// Mitsubishi GX Works2 project: BookEX3_2 FB   PLC: Q13UDV

TYPE DateTime : STRUCT
  Year : INT;
  Month : INT;
  Day : INT;
  WeekDay : INT;
  iHour : INT;
  iMin : INT;
  iSec : INT;
  ms : INT;
END_STRUCT END_TYPE

TYPE Vector : STRUCT
  axisX : REAL;
  axisY : REAL;
  axisZ : REAL;
END_STRUCT END_TYPE

TYPE WordBit : STRUCT
  Data : DWORD;
  Flag : BOOL;
END_STRUCT END_TYPE

// global labels: Global
VAR_GLOBAL
  bVar0 AT M5000 : BOOL;
  abArray0 AT M5010 : ARRAY [0..49] OF BOOL;
  sStr0 AT D5000 : STRING[199];
  sStr1 AT D5100 : STRING[199];
  sStr2 AT D5200 : STRING[199];
  sStr3 AT D5300 : STRING[199];
  sStr4 AT D5400 : STRING[199];
  sStr5 AT D5500 : STRING[199];
  sStr6 AT D5600 : STRING[199];
  sStr7 AT D5700 : STRING[199];
  sStr8 AT D5800 : STRING[199];
  sStr9 AT D5900 : STRING[199];
  iVar0 AT D4500 : INT;
  iVar1 AT D4501 : INT;
  iVar2 AT D4502 : INT;
  iVar3 AT D4503 : INT;
  iVar4 AT D4504 : INT;
  iVar5 AT D4505 : INT;
  iVar6 AT D4506 : INT;
  iVar7 AT D4507 : INT;
  iVar8 AT D4508 : INT;
  iVar9 AT D4509 : INT;
  dVar0 AT D4510 : DINT;
  dVar1 AT D4512 : DINT;
  dVar2 AT D4514 : DINT;
  dVar3 AT D4516 : DINT;
  dVar4 AT D4518 : DINT;
  dVar5 AT D4520 : DINT;
  dVar6 AT D4522 : DINT;
  dVar7 AT D4524 : DINT;
  dVar8 AT D4526 : DINT;
  dVar9 AT D4528 : DINT;
  wVar0 AT D4530 : WORD;
  wVar1 AT D4531 : WORD;
  wVar2 AT D4532 : WORD;
  wVar3 AT D4533 : WORD;
  wVar4 AT D4534 : WORD;
  wVar5 AT D4535 : WORD;
  wVar6 AT D4536 : WORD;
  wVar7 AT D4537 : WORD;
  wVar8 AT D4538 : WORD;
  wVar9 AT D4539 : WORD;
  dwVar0 AT D4540 : DWORD;
  dwVar1 AT D4542 : DWORD;
  dwVar2 AT D4544 : DWORD;
  dwVar3 AT D4546 : DWORD;
  dwVar4 AT D4548 : DWORD;
  dwVar5 AT D4550 : DWORD;
  dwVar6 AT D4552 : DWORD;
  dwVar7 AT D4554 : DWORD;
  dwVar8 AT D4556 : DWORD;
  dwVar9 AT D4558 : DWORD;
  fsVar0 AT D4560 : REAL;
  fsVar1 AT D4562 : REAL;
  fsVar2 AT D4564 : REAL;
  fsVar3 AT D4566 : REAL;
  fsVar4 AT D4568 : REAL;
  fsVar5 AT D4570 : REAL;
  fsVar6 AT D4572 : REAL;
  fsVar7 AT D4574 : REAL;
  fsVar8 AT D4576 : REAL;
  fsVar9 AT D4578 : REAL;
  fdVar0 AT D4580 : LREAL;
  tTime0 AT D4620 : TIME;
  tTime1 AT D4622 : TIME;
  tTime2 AT D4624 : TIME;
  tTime3 AT D4626 : TIME;
  tTime4 AT D4628 : TIME;
  tTime5 AT D4630 : TIME;
  tTime6 AT D4632 : TIME;
  tTime7 AT D4634 : TIME;
  tTime8 AT D4636 : TIME;
  tTime9 AT D4638 : TIME;
  tTime10 AT D4640 : TIME;
  bVar1 AT M5001 : BOOL;
  bVar2 AT M5002 : BOOL;
  bVar3 AT M5003 : BOOL;
  bVar4 AT M5004 : BOOL;
  bVar5 AT M5005 : BOOL;
  bVar6 AT M5006 : BOOL;
  bVar7 AT M5007 : BOOL;
  bVar8 AT M5008 : BOOL;
  bVar9 AT M5009 : BOOL;
  abArray1 AT M5060 : ARRAY [0..49] OF BOOL;
  abArray2 AT M5110 : ARRAY [0..49] OF BOOL;
  abArray3 AT M5160 : ARRAY [0..49] OF BOOL;
  abArray4 AT M5210 : ARRAY [0..49] OF BOOL;
  abArray5 AT M5260 : ARRAY [0..49] OF BOOL;
  abArray6 AT M5310 : ARRAY [0..49] OF BOOL;
  abArray7 AT M5360 : ARRAY [0..49] OF BOOL;
  abArray8 AT M5410 : ARRAY [0..49] OF BOOL;
  abArray9 AT M5460 : ARRAY [0..49] OF BOOL;
  fdVar1 AT D4584 : LREAL;
  fdVar2 AT D4588 : LREAL;
  fdVar3 AT D4592 : LREAL;
  fdVar4 AT D4596 : LREAL;
  fdVar5 AT D4600 : LREAL;
  fdVar6 AT D4604 : LREAL;
  fdVar7 AT D4608 : LREAL;
  fdVar8 AT D4612 : LREAL;
  fdVar9 AT D4616 : LREAL;
  afsPen0 AT D2000 : ARRAY [0..499] OF REAL;
  afsPen1 AT D3000 : ARRAY [0..499] OF REAL;
END_VAR
// user libraries (not included): HMI

FUNCTION_BLOCK UserFB
VAR_INPUT
  i_A : INT;
  i_B : INT;
END_VAR
VAR_OUTPUT
  i_C : INT;
END_VAR
;
i_C := i_A+i_B;
END_FUNCTION_BLOCK

FUNCTION_BLOCK UserFB_EN
VAR_INPUT
  i_A : INT;
  i_B : INT;
END_VAR
VAR_OUTPUT
  i_C : INT;
END_VAR
VAR_INPUT
  b_EN : BOOL;
END_VAR
VAR_OUTPUT
  b_ENO : BOOL;
END_VAR
;
b_ENO := b_EN;
IF NOT b_EN THEN
	RETURN;
END_IF;
i_C := i_A+i_B;
END_FUNCTION_BLOCK

FUNCTION_BLOCK UserFB_EN2
VAR_INPUT
  i_A : INT;
  i_B : INT;
END_VAR
VAR_OUTPUT
  i_C : INT;
END_VAR
VAR_INPUT
  b_EN : BOOL;
END_VAR
VAR_OUTPUT
  b_ENO : BOOL;
END_VAR
;
b_ENO := b_EN;
IF NOT b_EN THEN
	RETURN;
END_IF;
i_C := i_A+i_B;
END_FUNCTION_BLOCK

FUNCTION_BLOCK UserFBE
VAR_INPUT
  i_A : INT;
  i_B : INT;
END_VAR
VAR_OUTPUT
  i_C : INT;
END_VAR
;
i_C := i_A+i_B;
END_FUNCTION_BLOCK

FUNCTION_BLOCK UserFBE2
VAR_INPUT
  i_A : INT;
  i_B : INT;
END_VAR
VAR_OUTPUT
  i_C : INT;
END_VAR
;
i_C := i_A+i_B;
END_FUNCTION_BLOCK

FUNCTION UserFun
VAR_INPUT
  i_A : INT;
  i_B : INT;
END_VAR
;
UserFun := i_A+i_B;
END_FUNCTION

FUNCTION UserFunE
VAR_INPUT
  i_A : INT;
  i_B : INT;
END_VAR
;
UserFunE := i_A+i_B;
END_FUNCTION

PROGRAM ExEN_ENO
VAR
  UserFB_1 : UserFB;
  UserFBE_1 : UserFBE;
  UserFB_EN_1 : UserFB_EN;
  Mov4WORD_1 : Mov4WORD;
  UserFB_EN_2 : UserFB_EN;
  UserFBE2_1 : UserFBE2;
  UserFBE2_2 : UserFBE2;
  UserFB_EN2_1 : UserFB_EN2;
  UserFBE_3 : UserFBE;
  UserFBE2_3 : UserFBE2;
  UserFB_EN_3 : UserFB_EN;
  UserFB_EN2_2 : UserFB_EN2;
END_VAR
(* structured ladder/FBD written out as ST: instructions are called as NAME(EN, inputs, outputs); _pN, _eN, _tN stand for wires *)
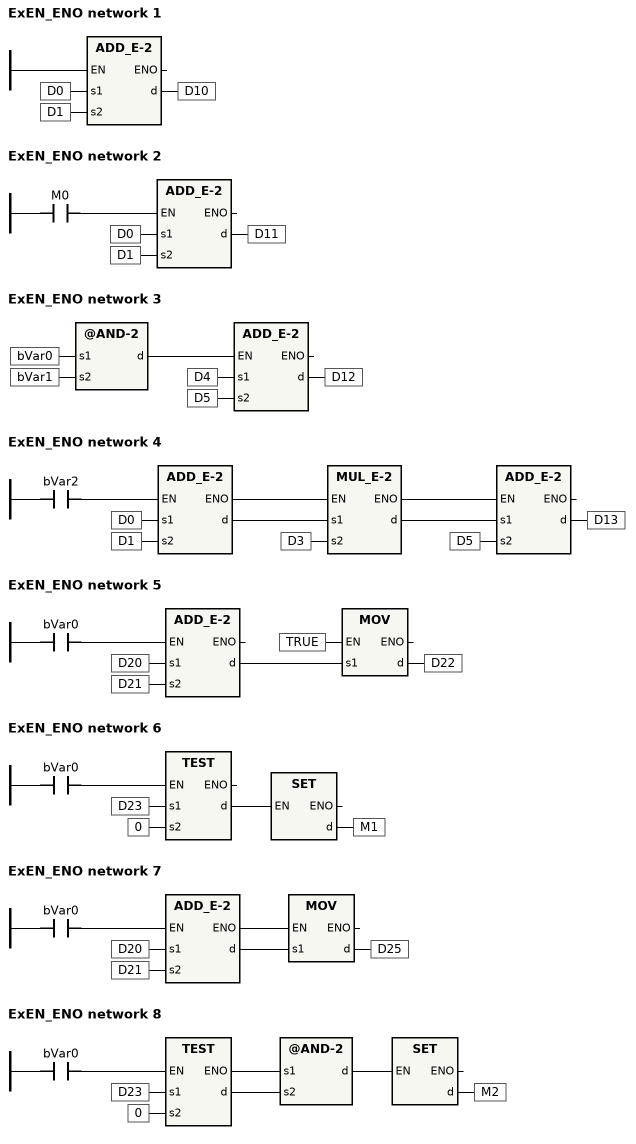
(* network 1 *)
ADD_E(TRUE, D0, D1, D10);
(* network 2 *)
ADD_E(M0, D0, D1, D11);
(* network 3 *)
ADD_E(@AND-2(bVar0, bVar1), D4, D5, D12);
(* network 4 *)
_e2 := ADD_E(bVar2, D0, D1, _t1);
_e4 := MUL_E(_e2, _t1, D3, _t3);
ADD_E(_e4, _t3, D5, D13);
(* network 5 *)
ADD_E(bVar0, D20, D21, _t1);
MOV(TRUE, _t1, D22);
(* network 6 *)
TEST(bVar0, D23, 0, _t1);
SET(_t1, M1);
(* network 7 *)
_e2 := ADD_E(bVar0, D20, D21, _t1);
MOV(_e2, _t1, D25);
(* network 8 *)
_e2 := TEST(bVar0, D23, 0, _t1);
SET(@AND-2(_e2, _t1), M2);
END_PROGRAM

PROGRAM ExFB
VAR
  TON_1 : TON;
  TON_E_1 : TON_E;
  R_TRIG_E_1 : R_TRIG_E;
  fbLabel_1 : fbLabel;
END_VAR
(* structured ladder/FBD written out as ST: instructions are called as NAME(EN, inputs, outputs); _pN, _eN, _tN stand for wires *)
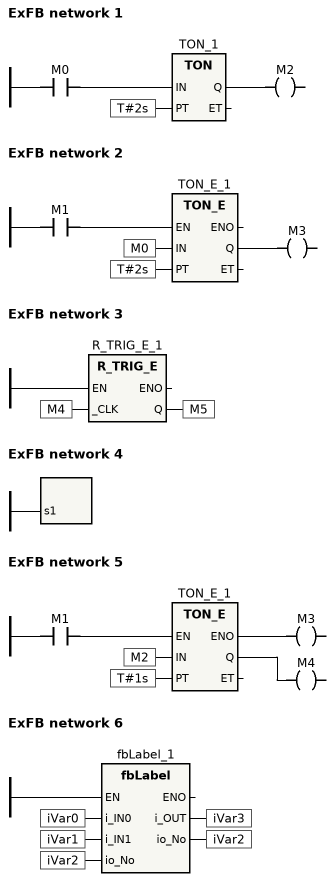
(* network 1 *)
TON_1(IN := M0, PT := T#2s);
M2 := TON_1.Q;
(* network 2 *)
TON_E_1(EN := M1, IN := M0, PT := T#2s);
M3 := TON_E_1.Q;
(* network 3 *)
R_TRIG_E_1(EN := TRUE, _CLK := M4, Q => M5);
(* network 4 *)
(* element kind 10  <- TRUE *)
(* network 5 *)
TON_E_1(EN := M1, IN := M2, PT := T#1s);
M3 := TON_E_1.ENO;
M4 := TON_E_1.Q;
(* network 6 *)
fbLabel_1(EN := TRUE, i_IN0 := iVar0, i_IN1 := iVar1, io_No := iVar2, i_OUT => iVar3);
iVar2 := fbLabel_1.io_No;
END_PROGRAM

PROGRAM ExFUN
(* structured ladder/FBD written out as ST: instructions are called as NAME(EN, inputs, outputs); _pN, _eN, _tN stand for wires *)
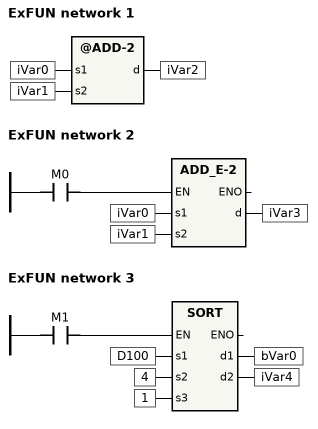
(* network 1 *)
iVar2 := @ADD-2(iVar0, iVar1);
(* network 2 *)
ADD_E(M0, iVar0, iVar1, iVar3);
(* network 3 *)
SORT(M1, D100, 4, 1, bVar0, iVar4);
END_PROGRAM

PROGRAM ExZR
(* structured ladder/FBD written out as ST: instructions are called as NAME(EN, inputs, outputs); _pN, _eN, _tN stand for wires *)
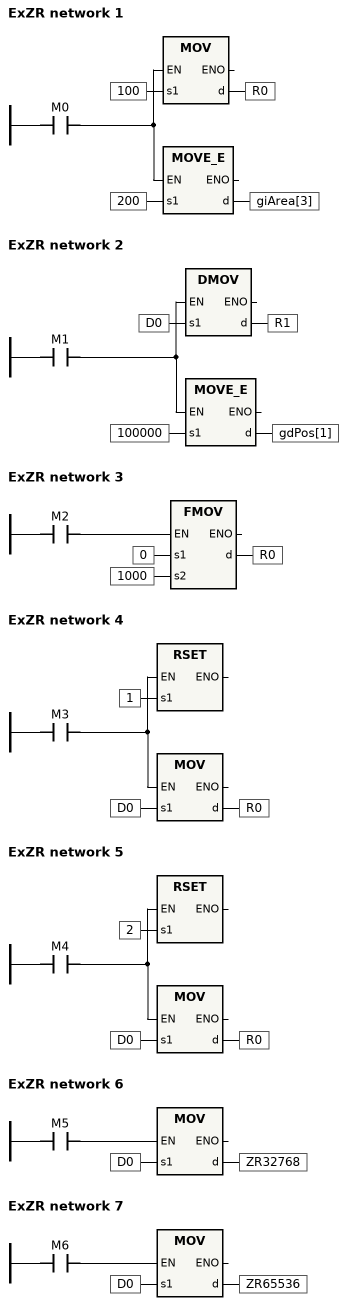
(* network 1 *)
MOV(M0, 100, R0);
MOVE_E(M0, 200, giArea[3]);
(* network 2 *)
DMOV(M1, D0, R1);
MOVE_E(M1, 100000, gdPos[1]);
(* network 3 *)
FMOV(M2, 0, 1000, R0);
(* network 4 *)
RSET(M3, 1);
MOV(M3, D0, R0);
(* network 5 *)
RSET(M4, 2);
MOV(M4, D0, R0);
(* network 6 *)
MOV(M5, D0, ZR32768);
(* network 7 *)
MOV(M6, D0, ZR65536);
END_PROGRAM

PROGRAM ExEN_ENO2
VAR
  UserFB_1 : UserFB;
  UserFBE_1 : UserFBE;
  UserFB_EN_1 : UserFB_EN;
  Mov4WORD_1 : Mov4WORD;
  UserFB_EN_2 : UserFB_EN;
  UserFBE2_1 : UserFBE2;
  UserFBE2_2 : UserFBE2;
  UserFB_EN2_1 : UserFB_EN2;
  UserFBE_3 : UserFBE;
  UserFBE2_3 : UserFBE2;
  UserFB_EN_3 : UserFB_EN;
  UserFB_EN2_2 : UserFB_EN2;
  UserFBE3_1 : UserFBE3;
END_VAR
(* structured ladder/FBD written out as ST: instructions are called as NAME(EN, inputs, outputs); _pN, _eN, _tN stand for wires *)
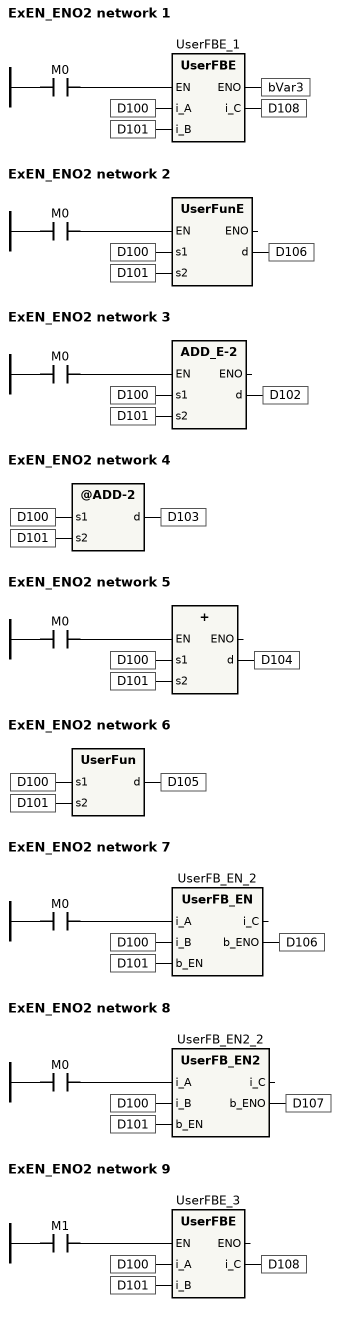
(* network 1 *)
UserFBE_1(EN := M0, i_A := D100, i_B := D101, ENO => bVar3, i_C => D108);
(* network 2 *)
UserFunE(M0, D100, D101, D106);
(* network 3 *)
ADD_E(M0, D100, D101, D102);
(* network 4 *)
D103 := @ADD-2(D100, D101);
(* network 5 *)
+(M0, D100, D101, D104);
(* network 6 *)
D105 := UserFun(D100, D101);
(* network 7 *)
UserFB_EN_2(i_A := M0, i_B := D100, b_EN := D101, b_ENO => D106);
(* network 8 *)
UserFB_EN2_2(i_A := M0, i_B := D100, b_EN := D101, b_ENO => D107);
(* network 9 *)
UserFBE_3(EN := M1, i_A := D100, i_B := D101, i_C => D108);
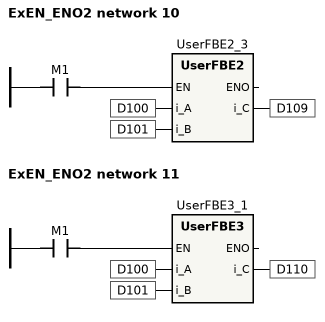
(* network 10 *)
UserFBE2_3(EN := M1, i_A := D100, i_B := D101, i_C => D109);
(* network 11 *)
UserFBE3_1(EN := M1, i_A := D100, i_B := D101, i_C => D110);
END_PROGRAM

FUNCTION_BLOCK UserFBE3
VAR_INPUT
  i_A : INT;
  i_B : INT;
END_VAR
VAR_OUTPUT
  i_C : INT;
END_VAR
;
i_C := i_A+i_B;
END_FUNCTION_BLOCK

FUNCTION_BLOCK fbLabel
VAR_INPUT
  i_IN0 : INT;
  i_IN1 : INT;
END_VAR
VAR_OUTPUT
  i_OUT : INT;
END_VAR
VAR_IN_OUT
  io_No : INT;
END_VAR
VAR
  ix : INT;
END_VAR
END_FUNCTION_BLOCK
